# EPICS substitutions: odmApp/Db/odm-sys0-od02.substitutions
file bkh_odm_common.db {
pattern
    {            P,     M,       LOC}
    {BKH:LI00:OD01, BKH01, L2KA01-08}
    {BKH:LI01:OD01, BKH02, L2KA01-08}
    {BKH:LI02:OD01, BKH03, L2KA02-09}
    {BKH:LI03:OD01, BKH04, L2KA03-07}
    {BKH:LI04:OD01, BKH05, L2KA04-06}
    {BKH:LI05:OD01, BKH06, L2KA05-07}
    {BKH:LI06:OD01, BKH07, L2KA06-08}
    {BKH:LI07:OD01, BKH08, L2KA07-03}
}

file bkh_odm_supervisor.db {
pattern
    {            P,     M,       LOC}
    {BKH:LI03:OD02, BKH09, L2KA03-07}
}

# Conversions --------------------------------
# Sensor cell monitors
file ai_convert_autosave.template {
pattern
    {                          INPV,                OUTPV,                   DESC,    C0,    C1, EGU, PREC, LOLO,  LOW, HIGH, HIHI,     LLSV,      LSV,      HSV,     HHSV}
    {"BKH:LI01:OD01:3012_01_CH01_I", "ODM:LI01:1:Cell:O2", "Sector 01, Sensor 01",  -7.5, 1.875, "%",    1, 19.0, 20.0, 23.0, 24.0, NO_ALARM, NO_ALARM, NO_ALARM, NO_ALARM}
    {"BKH:LI01:OD01:3012_01_CH02_I", "ODM:LI01:2:Cell:O2", "Sector 01, Sensor 02",  -7.5, 1.875, "%",    1, 19.0, 20.0, 23.0, 24.0, NO_ALARM, NO_ALARM, NO_ALARM, NO_ALARM}
    {"BKH:LI02:OD01:3012_01_CH01_I", "ODM:LI02:1:Cell:O2", "Sector 02, Sensor 01",  -7.5, 1.875, "%",    1, 19.0, 20.0, 23.0, 24.0, NO_ALARM, NO_ALARM, NO_ALARM, NO_ALARM}
    {"BKH:LI02:OD01:3012_01_CH02_I", "ODM:LI02:2:Cell:O2", "Sector 02, Sensor 02",  -7.5, 1.875, "%",    1, 19.0, 20.0, 23.0, 24.0, NO_ALARM, NO_ALARM, NO_ALARM, NO_ALARM}
    {"BKH:LI03:OD01:3012_01_CH01_I", "ODM:LI03:1:Cell:O2", "Sector 03, Sensor 01",  -7.5, 1.875, "%",    1, 19.0, 20.0, 23.0, 24.0, NO_ALARM, NO_ALARM, NO_ALARM, NO_ALARM}
    {"BKH:LI04:OD01:3012_01_CH01_I", "ODM:LI04:1:Cell:O2", "Sector 04, Sensor 01",  -7.5, 1.875, "%",    1, 19.0, 20.0, 23.0, 24.0, NO_ALARM, NO_ALARM, NO_ALARM, NO_ALARM}
    {"BKH:LI04:OD01:3012_01_CH02_I", "ODM:LI04:2:Cell:O2", "Sector 04, Sensor 02",  -7.5, 1.875, "%",    1, 19.0, 20.0, 23.0, 24.0, NO_ALARM, NO_ALARM, NO_ALARM, NO_ALARM}
    {"BKH:LI05:OD01:3012_01_CH01_I", "ODM:LI05:1:Cell:O2", "Sector 05, Sensor 01",  -7.5, 1.875, "%",    1, 19.0, 20.0, 23.0, 24.0, NO_ALARM, NO_ALARM, NO_ALARM, NO_ALARM}
    {"BKH:LI06:OD01:3012_01_CH01_I", "ODM:LI06:1:Cell:O2", "Sector 06, Sensor 01",  -7.5, 1.875, "%",    1, 19.0, 20.0, 23.0, 24.0, NO_ALARM, NO_ALARM, NO_ALARM, NO_ALARM}
    {"BKH:LI07:OD01:3012_01_CH01_I", "ODM:LI07:1:Cell:O2", "Sector 07, Sensor 01",  -7.5, 1.875, "%",    1, 19.0, 20.0, 23.0, 24.0, NO_ALARM, NO_ALARM, NO_ALARM, NO_ALARM}
}

# Supervisor
file bi_convert.template {
pattern
    {                           INPV,                          OUTPV,                           DESC,    ZNAM,  ONAM,      ZSV,      OSV}
    {"BKH:LI03:OD02:1104_01_CH01 MS",  "ODM:LI00:OD02:L1AlarmStatus", "Sec 00, Level-1 Tunnel Alarm", NoAlarm, Alarm, NO_ALARM,    MAJOR}
    {"BKH:LI03:OD02:1104_01_CH02 MS",  "ODM:LI00:OD02:L2AlarmStatus", "Sec 00, Level-2 Tunnel Alarm", NoAlarm, Alarm, NO_ALARM,    MAJOR}
    {"BKH:LI03:OD02:1104_01_CH03 MS",  "ODM:LI01:OD02:L1AlarmStatus", "Sec 01, Level-1 Tunnel Alarm", NoAlarm, Alarm, NO_ALARM,    MAJOR}
    {"BKH:LI03:OD02:1104_01_CH04 MS",  "ODM:LI01:OD02:L2AlarmStatus", "Sec 01, Level-2 Tunnel Alarm", NoAlarm, Alarm, NO_ALARM,    MAJOR}
    {"BKH:LI03:OD02:1104_01_CH05 MS",  "ODM:LI02:OD02:L1AlarmStatus", "Sec 02, Level-1 Tunnel Alarm", NoAlarm, Alarm, NO_ALARM,    MAJOR}
    {"BKH:LI03:OD02:1104_01_CH06 MS",  "ODM:LI02:OD02:L2AlarmStatus", "Sec 02, Level-2 Tunnel Alarm", NoAlarm, Alarm, NO_ALARM,    MAJOR}
    {"BKH:LI03:OD02:1104_01_CH07 MS",  "ODM:LI03:OD02:L1AlarmStatus", "Sec 03, Level-1 Tunnel Alarm", NoAlarm, Alarm, NO_ALARM,    MAJOR}
    {"BKH:LI03:OD02:1104_01_CH08 MS",  "ODM:LI03:OD02:L2AlarmStatus", "Sec 03, Level-2 Tunnel Alarm", NoAlarm, Alarm, NO_ALARM,    MAJOR}
    {"BKH:LI03:OD02:1104_01_CH09 MS",  "ODM:LI04:OD02:L1AlarmStatus", "Sec 04, Level-1 Tunnel Alarm", NoAlarm, Alarm, NO_ALARM,    MAJOR}
    {"BKH:LI03:OD02:1104_01_CH10 MS",  "ODM:LI04:OD02:L2AlarmStatus", "Sec 04, Level-2 Tunnel Alarm", NoAlarm, Alarm, NO_ALARM,    MAJOR}
    {"BKH:LI03:OD02:1104_01_CH11 MS",  "ODM:LI05:OD02:L1AlarmStatus", "Sec 05, Level-1 Tunnel Alarm", NoAlarm, Alarm, NO_ALARM,    MAJOR}
    {"BKH:LI03:OD02:1104_01_CH12 MS",  "ODM:LI05:OD02:L2AlarmStatus", "Sec 05, Level-2 Tunnel Alarm", NoAlarm, Alarm, NO_ALARM,    MAJOR}
    {"BKH:LI03:OD02:1104_01_CH13 MS",  "ODM:LI06:OD02:L1AlarmStatus", "Sec 06, Level-1 Tunnel Alarm", NoAlarm, Alarm, NO_ALARM,    MAJOR}
    {"BKH:LI03:OD02:1104_01_CH14 MS",  "ODM:LI06:OD02:L2AlarmStatus", "Sec 06, Level-2 Tunnel Alarm", NoAlarm, Alarm, NO_ALARM,    MAJOR}
    {"BKH:LI03:OD02:1104_01_CH15 MS",  "ODM:LI07:OD02:L1AlarmStatus", "Sec 07, Level-1 Tunnel Alarm", NoAlarm, Alarm, NO_ALARM,    MAJOR}
    {"BKH:LI03:OD02:1104_01_CH16 MS",  "ODM:LI07:OD02:L2AlarmStatus", "Sec 07, Level-2 Tunnel Alarm", NoAlarm, Alarm, NO_ALARM,    MAJOR}
    {"BKH:LI03:OD02:1104_01_CH17 MS",  "ODM:SYS0:OD02:SuprHrtbtAlarm","Supervisor HB Alarm Summary", NoAlarm, Alarm, NO_ALARM,    MAJOR}
    {"BKH:LI03:OD02:1104_01_CH18 MS",  "ODM:SYS0:OD02:SuprHrtbt",     "Supervisor Heartbeat",     Off,    On, NO_ALARM, NO_ALARM}
    {"BKH:LI03:OD02:1104_01_CH21 MS",  "ODM:LI00:OD02:PilzHBAlarm",   "Pilz Heartbeat Alarm S00", NoAlarm, Alarm, NO_ALARM,    MAJOR}
    {"BKH:LI03:OD02:1104_01_CH22 MS",  "ODM:LI01:OD02:PilzHBAlarm",   "Pilz Heartbeat Alarm S01", NoAlarm, Alarm, NO_ALARM,    MAJOR}
    {"BKH:LI03:OD02:1104_01_CH23 MS",  "ODM:LI02:OD02:PilzHBAlarm",   "Pilz Heartbeat Alarm S02", NoAlarm, Alarm, NO_ALARM,    MAJOR}
    {"BKH:LI03:OD02:1104_01_CH24 MS",  "ODM:LI03:OD02:PilzHBAlarm",   "Pilz Heartbeat Alarm S03", NoAlarm, Alarm, NO_ALARM,    MAJOR}
    {"BKH:LI03:OD02:1104_01_CH25 MS",  "ODM:LI04:OD02:PilzHBAlarm",   "Pilz Heartbeat Alarm S04", NoAlarm, Alarm, NO_ALARM,    MAJOR}
    {"BKH:LI03:OD02:1104_01_CH26 MS",  "ODM:LI05:OD02:PilzHBAlarm",   "Pilz Heartbeat Alarm S05", NoAlarm, Alarm, NO_ALARM,    MAJOR}
    {"BKH:LI03:OD02:1104_01_CH27 MS",  "ODM:LI06:OD02:PilzHBAlarm",   "Pilz Heartbeat Alarm S06", NoAlarm, Alarm, NO_ALARM,    MAJOR}
    {"BKH:LI03:OD02:1104_01_CH28 MS",  "ODM:LI07:OD02:PilzHBAlarm",   "Pilz Heartbeat Alarm S07", NoAlarm, Alarm, NO_ALARM,    MAJOR}
    {"BKH:LI03:OD02:1104_01_CH29 MS",  "ODM:LI08:OD02:L1AlarmStatus", "Sec 08, Level-1 Tunnel Alarm", NoAlarm, Alarm, NO_ALARM,    MAJOR}
    {"BKH:LI03:OD02:1104_01_CH30 MS",  "ODM:LI08:OD02:L2AlarmStatus", "Sec 08, Level-2 Tunnel Alarm", NoAlarm, Alarm, NO_ALARM,    MAJOR}
    {"BKH:LI03:OD02:1104_01_CH31 MS",  "ODM:LI09:OD02:L1AlarmStatus", "Sec 09, Level-1 Tunnel Alarm", NoAlarm, Alarm, NO_ALARM,    MAJOR}
    {"BKH:LI03:OD02:1104_01_CH32 MS",  "ODM:LI09:OD02:L2AlarmStatus", "Sec 09, Level-2 Tunnel Alarm", NoAlarm, Alarm, NO_ALARM,    MAJOR}
    {"BKH:LI03:OD02:1104_01_CH33 MS",  "ODM:LI10:OD02:L1AlarmStatus", "Sec 10, Level-1 Tunnel Alarm", NoAlarm, Alarm, NO_ALARM,    MAJOR}
    {"BKH:LI03:OD02:1104_01_CH34 MS",  "ODM:LI10:OD02:L2AlarmStatus", "Sec 10, Level-2 Tunnel Alarm", NoAlarm, Alarm, NO_ALARM,    MAJOR}
}

# Supervisor
file bo_convert.template {
pattern
    {                       OUTPV,                              INPV,                    DESC,    ZNAM,  ONAM, HIGH}
    {"BKH:LI03:OD02:2114_01_CH01", "ODM:SYS0:OD02:SuprHrtbtAlmReset", "Heartbeat Alarm Reset", Standby, Reset, 0.25}
}
